(* CODESYS project 02_FileWriteOnSDCardWithVisu.ecp

Project tree, tasks and I/O mapping:
  PFC200 : 750-8212 PFC200 G2 2ETH RS, WAGO, order no. 0750-8212, version 5.16.3.16
    application Application
      libraries: WagoAppTime, 1.7.3.3 (WAGO); WagoAppFileDir, 1.6.2.1 (WAGO)
      task PLC_Task (cyclic, interval 50 ms, priority 15) calls PLC_PRG
      task VISU_TASK (cyclic, interval 100 ms, priority 15) calls VisuElems.Visu_Prg
      task taskSchreibeDatei (cyclic, interval t#10ms, priority 15) calls prgWriteFile
      program PLC_PRG [ST]
      data type typMachineData
      data type typReal2Word
      visualisation Visualization
      program prgWriteFile [ST]
      global variables GVL
    ProjectConfiguration
    Kbus : Kbus, WAGO, version 1.4.0.2
        unmapped channels: K-BUS diagnostics
    MODBUS
      MODBUS : MODBUS, WAGO, order no. n/a, version 1.1.1.16
    Serial
      COM1 : COM1, WAGO, version 0.0.0.19
    Common.PCI
    EtherNet/IP
      Ethernet : Ethernet, WAGO, version 35.16.0.0
  libraries: VisuSymbols, 3.5.10.0 (System); WagoVisuIcons, 1.1.0.3 (WAGO)
  text list GlobalTextList
  00000000-0000-0000-0000-000000000000|C:\Users\u0100068\AppData\Local\Temp\1103d03de5bc4a0a8dba3d40d1b87c13\e868b832187f4f1a859da50215710801\Project.xml
*)

// PFC200/Application/typMachineData
TYPE typMachineData :
STRUCT
	sRange:			STRING(32);				// e.g. soldering machine 
	rCurrentL1, rCurrentL2, rCurrentL3: REAL;		// A
	rHeatDemand:	REAL;					// kWh
	sTimeStamp:		STRING(8);				// hh:mm
	dwStatus:		DWORD;					// 32 Boolean signals
											// single booleans are unefficient, eight bit for 1 bool variable is needed 
END_STRUCT
END_TYPE

// PFC200/Application/typReal2Word
TYPE typReal2Word :
UNION
	rData:	REAL;					// REAL
	awData:	ARRAY[0..1] OF WORD;	// 2 WORDs
	abData:	ARRAY[0..3] OF BYTE;	// 4 BYTEs
END_UNION
END_TYPE

// PFC200/Application/GVL
{attribute 'qualified_only'}
VAR_GLOBAL
	xTrigger:		BOOL;
	sOneDataset:	MaxString;
END_VAR

// PFC200/Application/PLC_PRG
PROGRAM PLC_PRG
VAR
	stDateTime:		WagoTypes.typWagoTimeComponents;
	sDateTime:		STRING(20);
	sTimeStamp:		STRING(8);
	i, j:			INT;						// shift F2 ==> reopen variable declaration
	trgMinute:		R_TRIG;
	// macine data acquisition
	astMachineData:	ARRAY[0..1439] OF typMachineData;
	uThermokon:		typReal2Word;
	uiRemainingTime: UINT;	
	iTemp01Raw:		INT := 345;
	wIn01:			WORD := 12345;
END_VAR

// CTRL space ==> intellisense

// get date and time
stDateTime := WagoAppTime.FuGetLocalTimeComponents();

// format a string, German date time format
sDateTime := WagoAppString.Format6(
	sFormat	:= '%02i.%02i.%4i %02i:%02i:%02i',
//	sFormat	:= '%4i/%02i/%02i %02i:%02i:%02i',	// England
	p1		:= ADR(stDateTime.uiDay),
	p2		:= ADR(stDateTime.uiMonth),
	p3		:= ADR(stDateTime.uiYear),
	p4		:= ADR(stDateTime.uiHour),
	p5		:= ADR(stDateTime.uiMinute),
	p6		:= ADR(stDateTime.uiSecond));

// format just hours and minutes
sTimeStamp := WagoAppString.Format2(
	sFormat	:= '%02i:%02i',
	p1		:= ADR(stDateTime.uiHour),
	p2		:= ADR(stDateTime.uiMinute));

// trigger every time, the minute gets zero
trgMinute(CLK := stDateTime.uiSecond = 0);
IF trgMinute.Q THEN
	// better use an averaging here (deutsch: Mittelwertbildung)
	// every minute we capture a complete dataset
	// the index consists of hour and minute
	j := TO_INT(stDateTime.uiHour * 60 + stDateTime.uiMinute);
	astMachineData[j].sRange := 'Hall of the mountain king';
	// these are just some changing values
	astMachineData[j].rCurrentL1 := 12.34 + iTemp01Raw / 12.34;
	astMachineData[j].rCurrentL2 := 12.34 + iTemp01Raw / 14.34;
	astMachineData[j].rCurrentL3 := 12.34 + iTemp01Raw / 11.34;
	astMachineData[j].rHeatDemand := 14.4 + iTemp01Raw * 1.2;
	astMachineData[j].sTimeStamp := sTimeStamp;
	astMachineData[j].dwStatus := wIn01;
	// combine the single values to one string and add carriage return and line feed
	GVL.sOneDataset := Format7(
		sFormat	:= '%s; %5.2f; %5.2f; %5.2f; %7.2f; %s; %i$R$N',
		p1:= ADR(astMachineData[j].sRange),
		p2:= ADR(astMachineData[j].rCurrentL1),
		p3:= ADR(astMachineData[j].rCurrentL2),
		p4:= ADR(astMachineData[j].rCurrentL3),
		p5:= ADR(astMachineData[j].rHeatDemand),
		p6:= ADR(astMachineData[j].sTimeStamp),
		p7:= ADR(astMachineData[j].dwStatus));
	// write dataset, see prgWriteFile
	GVL.xTrigger := TRUE;
END_IF
uiRemainingTime := 60 - stDateTime.uiSecond;

END_PROGRAM

// PFC200/Application/prgWriteFile
PROGRAM prgWriteFile
VAR
	fbFile:			WagoAppFileDir.FbGeneralFile;
	fbFileOpen:		WagoAppFileDir.FbGeneralFile_Open_mod;
	fbFileWrite:	WagoAppFileDir.FbGeneralFile_Write_mod;
	fbFileClose:	WagoAppFileDir.FbGeneralFile_Close_mod;
	xFileIsOpen, xFileIsWritten, xFileIsClosed: BOOL;
	// extension: the name of the file should be changed at the end of the day
	// at the moment the file will be overwritten each morning
	// only use this folder, when there's no sd card available
	sName:			STRING(30) := '/var/www/hurgahossa.csv';
	// path to the sd card
//	sName:			STRING(30) := '/media/sd/hurgahossa.csv';
END_VAR

// enhancement: check, if sd card is present with: FbCheckDirectoryExists

fbFileOpen(
	oStatus		=> ,
	xExecute	:= GVL.xTrigger,	// open the file when the trigger has been set
	xError		=> ,
	xDone		=> xFileIsOpen,		// tell me when the file is open
	xBusy		=> ,
	Instance	:= fbFile,
	xIsOpen		=> ,
	xEofReached	=> ,
	sName		:= sName,			// open the file with your browser: 192.168.1.xxx/hurgahossa.csv
	eAccMode	:= eFileAccessMode.FAM_Append,		// append data
	eSyncMode	:= eFileSyncMode.FSM_SafeClose,
	xExclusive	:= );

fbFileWrite(
	oStatus		=> ,
	xExecute	:= xFileIsOpen,		// write data when the file is open
	xError		=> ,
	xDone		=> xFileIsWritten,	// tell me when the data has been written
	xBusy		=> ,
	Instance	:= fbFile,
	xIsOpen		=> ,
	xEofReached	=> ,
	pTxBuffer	:= ADR(GVL.sOneDataset),			// write one dataset
	udiTxNBytes	:= TO_UDINT(LEN(STR := GVL.sOneDataset)));		// the length of one dataset

fbFileClose(
	oStatus		=> ,
	xExecute	:= xFileIsWritten,	// close the file when the data has been written
	xError		=> ,
	xDone		=> xFileIsClosed,	// tell me when the file has been closed
	xBusy		=> ,
	Instance	:= fbFile,
	xIsOpen		=> ,
	xEofReached	=> );

IF xFileIsClosed THEN
	GVL.xTrigger := FALSE;			// reset the trigger when the file has been closed 
END_IF;

END_PROGRAM

// PFC200/Application/Visualization
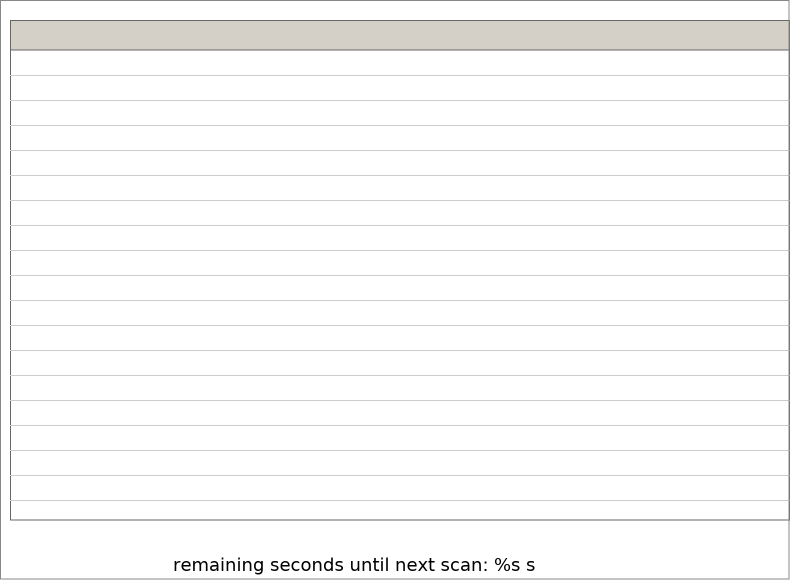
VISUALIZATION Visualization  // 790x580
    Table (10,20 780x500), data array: PLC_PRG.astMachineData
        p3854506369: PLC_PRG.astMachineData[INDEX].sRange
        p1892666644: PLC_PRG.astMachineData[INDEX].rCurrentL1
        p338671338: PLC_PRG.astMachineData[INDEX].rCurrentL2
        p2170511999: PLC_PRG.astMachineData[INDEX].rCurrentL3
        p3723444502: PLC_PRG.astMachineData[INDEX].rHeatDemand
        p1218418051: PLC_PRG.astMachineData[INDEX].sTimeStamp
        p746581629: PLC_PRG.astMachineData[INDEX].dwStatus
        p2232123230: range
        p511219082: current L1
        p1755163831: current L2
        p4092479075: current L3
        p2237128397: heat demand
        p505689113: time stamp
        p1757482276: status
        p1137915858: PLC_PRG.j
        p1014161805: 1439 - 0 + 1
    Textfield (170,550 390x30), "remaining seconds until next scan: %s s", text variable: PLC_PRG.uiRemainingTime
END_VISUALIZATION
